# EPICS StreamDevice protocol: protocols/sync_role.proto
Terminator = LF;
ExtraInput = Ignore;
ReplyTimeout = 4000;

set_sync_role {
	out "sync_role %s";
	in;
}

get_sync_role {
	out "sync_role";
	in "%40c";
}

get_sync_role_fs {
        out "sync_role_fs";
        in "%d";
}

setCounterLatch {
	out "counter_latch %d";
	in;
}
